FUNCTION_BLOCK FB_MotionAxisDS402NC IMPLEMENTS I_MotionAxis
VAR_INPUT
END_VAR
VAR_OUTPUT
END_VAR
VAR
    {attribute 'no_copy'}
    AxisRef : REFERENCE TO AXIS_REF;
    iMotionAxisCommon : I_MotionAxisCommon;
    // NC Blocks
    fbSetPos		:	MC_SetPosition;
     bClearPositionLag : BOOL := TRUE;

    // create a property for some of these
    bExecMove			: BOOL;
    bExecHome			: BOOL;
    bPosGoal			: BOOL;
    bNegGoal			: BOOL;
    bNewMoveReq			: BOOL;
    bHomingBusy			: BOOL;
    bHomingDone			: BOOL;
    bPrepareDisable		: BOOL;
    bMoveDone			: BOOL;
    bMoveBusy			: BOOL;
    bHalted				: BOOL;
    bAborted			: BOOL;
    bStopped			: BOOL;
    bOperational		: BOOL;
    bServoOffTrans		: BOOL;
    bServoOnTrans 		: BOOL;
    bServoOffMode		: BOOL ;
    bServoOnMode		: BOOL;
    bDiscreteInit		: BOOL;
    bDiscreteMotionAct  : BOOL;
    bServoOffparamsSet  : BOOL;
    bServoOffparamsSetDone : BOOL;
    bLimOverride				: BOOL;
    bPositionHolding		: BOOL;
    bError				: BOOL:=FALSE;
    bErrorStop			: BOOL;
    // use this for motion time axis states
    bExecute			: BOOL;
    // This prevent unexpected logical 1 on stMotionStage.bExecute
    nErrorId			: UDINT:=0;
    sLocalErrorMessage	: STRING;
    nPiezoErrorCode		: UDINT;
    // Save abd restore encoder value
    bInit				: BOOL;
    bLoad				: BOOL;
    bEncError			: BOOL;
    bSaveDone			: BOOL;
    bAbortDone			: BOOL;
    // axis status -- emulating some NC axis
    bClosedLoopMode		:	BOOL;
    bPositiveDirection	:  	BOOL;
    bNegativeDirection 	:  	BOOL;
    bInTargetPosition 	:  	BOOL;
    bReadErrDone			: 	BOOL;
    bLogReady			: 	BOOL;
    bFault				: 	BOOL;
    bDiscreteMotion 	:  	BOOL;
    bContinuousMotion 	:  	BOOL;
    bSlowParamReadTimer	: 	BOOL := TRUE;

    rtHaltedDone	: R_TRIG;
    rtTargetReached	: R_TRIG;
    ftAbortDone: F_TRIG;
    rtFault			: R_TRIG;
    rtHomed			: R_TRIG;
    rtMoveCmdShortcut	: R_TRIG;
    rtHomeCmdShortcut	: R_TRIG;
    rtEnableMode		: R_TRIG;
    rtUserExec			: R_TRIG;
    rtModeChange			: R_TRIG;
    rtTarget		: R_TRIG;
    rtServoOnMode	: R_TRIG;
    rtEnableDrive	: R_TRIG;
    rtServoOnTrans	: R_TRIG;
    rtNotClState 	: R_TRIG;
    rtNotOlState 	: R_TRIG;
    rtNewMoveReq	: R_TRIG;
    rtNewHoldTime	: R_TRIG;
    ftServoOffTrans	: F_TRIG;
    rtServoOffMode	: R_TRIG;
    ftAmsNetId 		: F_TRIG;
    ftExec			: F_TRIG;
    ftErrorSdoRead	: F_TRIG;
    ftEnableDrive	: F_TRIG;
    ftForwardEnabled	: F_TRIG;
    ftBackwardEnabled	: F_TRIG;
    ftServo				: F_TRIG;

    ftSdoStep		: 	F_TRIG;
    ftSdoStepFreq	: 	F_TRIG;
    ftSdoStepAmp	: 	F_TRIG;

    tonSyncHoming 		: TON;
    tonHoldTime			: TON;
    tonServoOffSync		: TON;
    tonSlowParamReadTimer: TON;
    // fast changing paramter timer -- wwe could have used PDO for this params
    // but the Piezo ESC have fixed PDO list.
    tonFastParamReadTimer: TON;
    //bInitiated	: BOOL;
    // Diagnotics data from the drive, mainly Error codes
    tRefreshDelay   : TIME := T#1S;
    nSavedholtime	: UDINT;
    tholtime		: TIME := T#10S;
    // Open Loop Operations
    fbSdoStep		: 	FB_EcCoESdoWrite;
    fbSdoStepFreq	: 	FB_EcCoESdoWrite;
    fbSdoStepAmp	: 	FB_EcCoESdoWrite;

    fbErrorSdoRead			: FB_EcCoESdoRead;
    fbFollowWinSdoRead		: FB_EcCoESdoRead;
    fbSoftLimMaxSdoRead		: FB_EcCoESdoRead;
    fbSoftLimMinSdoRead 	: FB_EcCoESdoRead;
    fbMotorloadSdoRead		: FB_EcCoESdoRead;
    fbGetAmsNetId			: FB_GetLocalAmsNetId;

    sAmsNetId 				: T_AmsNetId;
    nSubIndex  				: BYTE := 0;

      nChanFErrWinIdx		: WORD;
      nChanSoftwareLimIdx	: WORD;
      nChanMotorLoadIdx	: WORD;
    nChanErrorCodeIdx	: WORD;
    nChanOlStepIdx		: WORD;
    nChanOlStepFreqIdx	: WORD;
    nChanOlStepAmpIdx	: WORD;

// NC Exposed Parameters
    bCtrlEnablePosDiffControl     : WORD;
    bEncEnableSoftEndMaxControl   : WORD;
    bEncEnableSoftEndMinControl   : WORD;
    fAccelerationMax              : LREAL;
    fCtrlPosDiffMax               : LREAL;
    fCtrlPosDiffMaxTime           : LREAL;
    fDecelerationMax              : LREAL;
    fEncSoftEndMax                : LREAL;
    fEncSoftEndMin                : LREAL;
    fVeloMaximum                  : LREAL;
    fEncOffset               	  : LREAL;
    fEncScaleFactorInternal       : LREAL;
END_VAR


VAR CONSTANT

    nMotorLoadbase		: WORD := 16#200D;
    nSoftLimBase		: WORD := 16#200e;
    nHomeOffsetBase		: WORD := 16#607C;
    nHomingSpeedBase	: WORD := 16#6099;
    nhomingAccBase		: WORD := 16#609a;
    nErrorCodeBase		: WORD := 16#603f;
    nFErrWinBase		: WORD := 16#6065;
    nOlStepBase			: WORD := 16#2022;
    nOlStepAmpBase		: WORD := 16#2023;
    nOlStepFreqBase		: WORD := 16#2024;
    // this true for SmartAct MCS2 and E-727.
    nChanOfsBase		: WORD := 16#800;
    // DS 402 Motor encoder defective code : this is needed for save and restore.
    nEncErrorCode		: WORD := 16#7300;
END_VAR

{warning 'Add method implementation '}
METHOD CalibrateEncValue
END_METHOD

PROPERTY ControlWord : UINT
GET
END_GET
SET
END_SET
END_PROPERTY

METHOD CyclicCalls
END_METHOD

PROPERTY EncOffset : LREAL
GET
EncOffset := fEncOffset;
END_GET
SET
fEncOffset := EncOffset;
END_SET
END_PROPERTY

{warning 'Add method implementation '}
METHOD EncSaveRestore
END_METHOD

PROPERTY Error : BOOL
GET
Error := bError;
END_GET
SET
bError := Error;
END_SET
END_PROPERTY

PROPERTY ErrorCode : UDINT
GET
ErrorCode := nErrorId;
END_GET
SET
nErrorId := ErrorCode;
END_SET
END_PROPERTY

//FB_Init is always available implicitly and it is used primarily for initialization.
//The return value is not evaluated. For a specific influence, you can also declare the
//methods explicitly and provide additional code there with the standard initialization
//code. You can evaluate the return value.
METHOD FB_Init: BOOL
VAR_INPUT
    bInitRetains: BOOL; // TRUE: the retain variables are initialized (reset warm / reset cold)
    bInCopyCode: BOOL;  // TRUE: the instance will be copied to the copy code afterward (online change)
    AxisReference : REFERENCE TO AXIS_REF;
    //iMotionAxisCommon : I_MotionAxisCommon;
END_VAR
AxisRef REF= AxisReference;
//iMotionAxisCommon := iMotionAxisCommon;
END_METHOD

{warning 'Add method implementation '}
METHOD GearIn
END_METHOD

{warning 'Add method implementation '}
METHOD GearOut
END_METHOD

{warning 'Add method implementation '}
METHOD GetAxisRef : REFERENCE TO AXIS_REF
END_METHOD

{warning 'Add method implementation '}
METHOD GetPowerOverride : LREAL
END_METHOD

{warning 'Add method implementation '}
METHOD Halt
VAR_INPUT
    Deceleration	: LREAL := 0.0;
    Jerk	: LREAL := 0.0;
    BufferMode	: MC_BufferMode := .MC_BufferMode.MC_Aborting;
END_VAR
VAR_OUTPUT
    Done	: BOOL;
    Busy	: BOOL;
    Active	: BOOL;
    CommandAborted	: BOOL;
    Error	: BOOL;
    ErrorID	: UDINT;
    ErrorStr	: T_MaxString;
END_VAR
END_METHOD

{warning 'Add property implementation'}
PROPERTY HaltBusy : BOOL
GET
END_GET
END_PROPERTY

{warning 'Add property implementation'}
PROPERTY HaltDone : BOOL
GET
END_GET
END_PROPERTY

{warning 'Add property implementation'}
PROPERTY HaltError : BOOL
GET
END_GET
END_PROPERTY

{warning 'Add property implementation'}
PROPERTY HaltErrorID : UDINT
GET
END_GET
END_PROPERTY

METHOD Home
//
// tonSyncHoming(PT:=T#500MS);
// (* IMPORTANT: Homing options and parameters must be configured either via the COE online tab or via the service tool *)
// CASE eHomingState OF
//     E_DS402Homing.INIT_HOMING :;
// 		rtModeChange (CLK:=(THIS^.ModeOfOperationDisplay = E_DS402OpMode.HOMING));
//         IF rtModeChange.Q THEN
// 			tonSyncHoming.IN := TRUE;
//             stPiezoStage.nPiezoDriveControl.4:=TRUE;
//         END_IF
// 		IF tonSyncHoming.Q THEN
// 			eHomingState:=E_DS402Homing.HOMING_IN_PROGRESS;
// 		END_IF
//     E_DS402Homing.HOMING_IN_PROGRESS:
//         IF NOT stPiezoStage.stPiezoDriveStatus.TargetReached
//            AND NOT stPiezoStage.stPiezoDriveStatus.Bit13_OpModeSpecific THEN
//                 HomingBusy:=TRUE;
//                 HomeDone:=FALSE;
//
//         // Interrupted
//         ELSIF Stopped AND stPiezoStage.bHalt THEN
//             eHomingState:=E_DS402Homing.HOMING_INTERRUPTED;
//
// 		// Genral Motion error i.e Following error ?
// 		ELSIF stPiezoStage.stPiezoDriveStatus.Bit13_OpModeSpecific THEN
// 			eHomingState:=E_DS402Homing.HOMING_ERROR;
//
//         // Reached
//         ELSIF stPiezoStage.stPiezoDriveStatus.TargetReached
//             AND stPiezoStage.stPiezoDriveStatus.Bit12_OpModeSpecific
//             AND NOT stPiezoStage.stPiezoDriveStatus.Bit13_OpModeSpecific THEN
//             eHomingState:=E_DS402Homing.HOMING_ATTAINED;
//         END_IF
//
//
//     E_DS402Homing.HOMING_INTERRUPTED :;
//         HomingBusy:=FALSE;
//         HomeDone:=FALSE;
// 		Halted := TRUE;
// 		McAxisState:= MC_AxisStates.MC_AXISSTATE_STOPPING;
//
//     E_DS402Homing.HOMING_ATTAINED:;
//         HomingBusy:=FALSE;
// 		tonSyncHoming.IN := FALSE;
// 		tonHoldTime.IN := TRUE;
// 		eHomingState:=E_DS402Homing.HOMING_DONE;
//
//     E_DS402Homing.HOMING_DONE:;
// 		//prepare next move
// 		IF NOT THIS^.PositionHolding THEN
// 			HomeDone:=TRUE;
// 			stPiezoStage.fPosition:=0.0;
// 			fbSetPos.Position := stPiezoStage.fPosition;
// 			fbSetPos.Execute := HomeDone;
// 			IF fbSetPos.bError THEN
// 				eHomingState:=E_DS402Homing.HOMING_ERROR;
// 			ELSE
// 				IF (fbSetPos.bDone) THEN
// 					fbSetPos.Execute := FALSE;
// 				END_IF
// 			END_IF
// 			PositionHolding := TRUE;
// 			stPiezoStage.nPiezoDriveControl.4:=FALSE;
// 		END_IF
//
//
//     E_DS402Homing.HOMING_ERROR :;
// 		Error:= TRUE;
// 		HomeDone:=FALSE;
// 		HomingBusy:= FALSE;
// 		IF fbSetPos.nErrorId <> 0 THEN
// 		// set an Error flag home, homing actually does sdo read on ErrorCode object
// 			ErrorCode := fbSetPos.nErrorId;
// 		ELSE
// 			McAxisState:=MC_AxisStates.MC_AXISSTATE_ERRORSTOP;
// 		END_IF
//
// END_CASE
//
// fbSetPos.Options.ClearPositionLag:= bClearPositionLag;
// fbSetPos( Axis:= stPiezoStage.Axis  );
END_METHOD

{warning 'Add property implementation'}
PROPERTY HomeDone : BOOL
GET
END_GET
SET
END_SET
END_PROPERTY

{warning 'Add property implementation'}
PROPERTY HomingBusy : BOOL
GET
END_GET
SET
END_SET
END_PROPERTY

{warning 'Add property implementation'}
PROPERTY MeasuredAcceleration : LREAL
GET
END_GET
END_PROPERTY

{warning 'Add property implementation'}
PROPERTY MeasuredPosition : LREAL
GET
END_GET
END_PROPERTY

{warning 'Add property implementation'}
PROPERTY MeasuredVelocity : LREAL
GET
END_GET
END_PROPERTY

PROPERTY ModeOfOperation : BOOL
GET
END_GET
SET
END_SET
END_PROPERTY

PROPERTY ModeOfOperationDisplay : INT
GET
END_GET
SET
END_SET
END_PROPERTY

{warning 'Add method implementation '}
METHOD MoveAbsolute
VAR_INPUT
    Position	: LREAL;
    Velocity	: LREAL;
    Acceleration	: LREAL := 0.0;
    Deceleration	: LREAL := 0.0;
    Jerk	: LREAL := 0.0;
    BufferMode	: MC_BufferMode := .MC_BufferMode.MC_Aborting;
END_VAR
VAR_OUTPUT
    Done	: BOOL;
    Busy	: BOOL;
    Active	: BOOL;
    CommandAborted	: BOOL;
    Error	: BOOL;
    ErrorID	: UDINT;
    ErrorStr	: T_MaxString;
END_VAR
END_METHOD

{warning 'Add property implementation'}
PROPERTY MoveAbsoluteBusy : BOOL
GET
END_GET
END_PROPERTY

{warning 'Add property implementation'}
PROPERTY MoveAbsoluteDone : BOOL
GET
END_GET
END_PROPERTY

{warning 'Add property implementation'}
PROPERTY MoveAbsoluteError : BOOL
GET
END_GET
END_PROPERTY

{warning 'Add property implementation'}
PROPERTY MoveAbsoluteErrorID : UDINT
GET
END_GET
END_PROPERTY

{warning 'Add property implementation'}
PROPERTY MoveAbsoluteTargetAcceleration : LREAL
GET
END_GET
END_PROPERTY

{warning 'Add property implementation'}
PROPERTY MoveAbsoluteTargetDeceleration : LREAL
GET
END_GET
END_PROPERTY

{warning 'Add property implementation'}
PROPERTY MoveAbsoluteTargetJerk : LREAL
GET
END_GET
END_PROPERTY

{warning 'Add property implementation'}
PROPERTY MoveAbsoluteTargetPosition : LREAL
GET
END_GET
END_PROPERTY

{warning 'Add property implementation'}
PROPERTY MoveAbsoluteTargetVelocity : LREAL
GET
END_GET
END_PROPERTY

{warning 'Add property implementation'}
PROPERTY MoveBusy : BOOL
GET
END_GET
SET
END_SET
END_PROPERTY

{warning 'Add property implementation'}
PROPERTY MoveDone : BOOL
GET
END_GET
SET
END_SET
END_PROPERTY

{warning 'Add property implementation'}
PROPERTY NegativeMotionIsEnabled : BOOL
GET
END_GET
END_PROPERTY

PROPERTY PositionHolding : BOOL
GET
END_GET
SET
END_SET
END_PROPERTY

{warning 'Add property implementation'}
PROPERTY PositiveMotionIsEnabled : BOOL
GET
END_GET
END_PROPERTY

METHOD Power
VAR_INPUT
    Enable	: BOOL;
    Enable_Positive	: BOOL;
    Enable_Negative	: BOOL;
    (* in percent from 0 to 100 *)
    Override	: LREAL := 100.0;
    BufferMode	: MC_BufferMode := .MC_BufferMode.MC_Aborting;
END_VAR
VAR_OUTPUT
    Status	: BOOL;
    Busy	: BOOL;
    Active	: BOOL;
    Error	: BOOL;
    ErrorID	: UDINT;
    ErrorStr	: T_MaxString;
END_VAR
END_METHOD

{warning 'Add property implementation'}
PROPERTY PowerError : BOOL
GET
END_GET
END_PROPERTY

{warning 'Add property implementation'}
PROPERTY PowerErrorID : UDINT
GET
END_GET
END_PROPERTY

{warning 'Add property implementation'}
PROPERTY PowerIsEnabled : BOOL
GET
END_GET
END_PROPERTY

{warning 'Add property implementation'}
PROPERTY PowerOverride : LREAL
GET
END_GET
END_PROPERTY

PROPERTY PowerStatus : BOOL
GET
END_GET
END_PROPERTY

{warning 'Add method implementation '}
METHOD Reset
VAR_OUTPUT
    Done	: BOOL;
    Busy	: BOOL;
    Error	: BOOL;
    ErrorID	: UDINT;
    ErrorStr	: T_MaxString;
END_VAR
END_METHOD

{warning 'Add property implementation'}
PROPERTY SetpointAcceleration : LREAL
GET
END_GET
END_PROPERTY

{warning 'Add property implementation'}
PROPERTY SetpointJerk : LREAL
GET
END_GET
END_PROPERTY

{warning 'Add property implementation'}
PROPERTY SetpointPosition : LREAL
GET
END_GET
END_PROPERTY

{warning 'Add property implementation'}
PROPERTY SetpointVelocity : LREAL
GET
END_GET
END_PROPERTY

{warning 'Add method implementation '}
METHOD SetPowerOverride
VAR_INPUT
    (* in percent from 0 to 100 *)
    Override	: LREAL;
END_VAR
VAR_OUTPUT
    Status	: BOOL;
    Busy	: BOOL;
    Active	: BOOL;
    Error	: BOOL;
    ErrorID	: UDINT;
    ErrorStr	: T_MaxString;
END_VAR
END_METHOD

END_FUNCTION_BLOCK

(* stored: Version 1.1.0.1
   POU FB_MotionAxisDS402NC: Id {c65bcaa5-32c2-4ba1-a44e-f37d90d611d0}, SpecialFunc None
   Method CalibrateEncValue: Id {91970a26-c709-4b22-9267-b0d1667fe522}
   Property ControlWord: Id {2e23514f-1ff8-4e7d-ba07-c83a3406e12d}
   Get Get: Id {d1d98f73-4ffe-4c5e-ac5b-39dd2029d583}
   Set Set: Id {7fe4a318-1fd6-4879-9b09-7166eef3accc}
   Method CyclicCalls: Id {4817919d-5e20-4c69-8186-0bdf3efe567b}
   Property EncOffset: Id {eb27fba9-5a73-44b3-af11-96a7e15e3ee9}
   Get Get: Id {4f5f199f-c50e-4b22-b7ed-6508a6417ac4}
   Set Set: Id {f81e3843-bcab-4cad-9e8e-d6f853087f87}
   Method EncSaveRestore: Id {395cb6b1-30cf-4c08-973a-ea5683a4aacb}
   Property Error: Id {6591e605-cd47-41e1-b465-f220aaf35b56}
   Get Get: Id {83c61458-bc47-4a5e-a9b2-bc79b90aa45e}
   Set Set: Id {ced43cf6-7634-420d-9841-a2c3186f3ec9}
   Property ErrorCode: Id {e4677a0d-4413-43f2-9c1c-22656f92edde}
   Get Get: Id {dd065214-6bd8-4f8e-aaae-f102862fe903}
   Set Set: Id {a96e7f86-e0ce-40c9-b81e-a4857450ab14}
   Method FB_Init: Id {3c6b89cf-6335-421f-bc49-43ad02ddd5d0}
   Method GearIn: Id {f2f47c3c-7d99-4ce3-b227-d63c7dadbcd1}
   Method GearOut: Id {df7b12cb-8329-492b-be94-64270ee0b5d3}
   Method GetAxisRef: Id {4c207fcd-ec74-4a2e-ba86-459e92aca7f0}
   Method GetPowerOverride: Id {baaece9b-c9ed-489a-91a6-6084d0b1301b}
   Method Halt: Id {b6a8e12d-141b-4b04-b9a3-63a5a6a53059}
   Property HaltBusy: Id {6de0810c-191e-4226-bd42-c87c979bb175}
   Get Get: Id {d49b1f45-1fdf-4987-913a-622876a70ea8}
   Property HaltDone: Id {a8f5b39a-39b9-4a5b-ad34-4985140fd6f3}
   Get Get: Id {c7f2d09e-21b3-40ba-a673-33daea3f18eb}
   Property HaltError: Id {2768033b-365c-4b0f-930b-fb1bc259fcf2}
   Get Get: Id {4cba867e-6440-4471-83ba-4d04bff8bddf}
   Property HaltErrorID: Id {529176ba-5239-45de-acf8-647c49afbae5}
   Get Get: Id {628ea864-33f6-43f6-8f24-83692e88db69}
   Method Home: Id {70bd90c9-eebc-4f8a-a8ba-43919335ed26}
   Property HomeDone: Id {3f03d77b-7aea-46cf-b024-61ea35080b25}
   Get Get: Id {25d464c0-bb5a-4130-86d9-11dd9c72a9ce}
   Set Set: Id {e5508470-c502-4410-bb85-a928cda5c3a3}
   Property HomingBusy: Id {73613f6b-5360-47c4-a9ca-b2b51b8e5224}
   Get Get: Id {21f2fba0-7289-43ea-9a84-75045f357048}
   Set Set: Id {2c2e2af5-2fee-46fd-b099-50f87b0689fc}
   Property MeasuredAcceleration: Id {e265c786-9035-4ea9-82fe-efff9985ed1b}
   Get Get: Id {405282c6-1f48-4d0b-9ca0-a1359e4ad562}
   Property MeasuredPosition: Id {210ba193-d721-4b65-bd1d-f2c43e4f1098}
   Get Get: Id {ea0c0a20-155f-480f-b77a-543c70a9ce7c}
   Property MeasuredVelocity: Id {cc7e62a9-ad83-4971-a6af-2ec0a8bfdfc3}
   Get Get: Id {7e3270c1-6958-4385-8fe5-a7f14d3aeafc}
   Property ModeOfOperation: Id {875d8e8c-6833-41bc-9ba1-506b540ec8bd}
   Get Get: Id {56d86dbd-488d-4d81-8fba-585be7d2afb4}
   Set Set: Id {cb4afb24-f6a8-483d-9128-b2270706924c}
   Property ModeOfOperationDisplay: Id {025cb625-ad11-4c51-9d0f-d907911a35f1}
   Get Get: Id {246a8b29-e645-4a6c-ba23-adb92ac595af}
   Set Set: Id {66c00ddb-4deb-4f26-b4ae-ee600494a340}
   Method MoveAbsolute: Id {6b50c75c-030a-4b3c-9a0b-c342bc66e047}
   Property MoveAbsoluteBusy: Id {2cd6cbfa-43df-4b87-bc54-2038020ebf9b}
   Get Get: Id {b6e2b46f-30ca-4446-92b6-ee2b61e9f9b2}
   Property MoveAbsoluteDone: Id {943f432d-764c-4ecb-a2a2-cb12fcf0605e}
   Get Get: Id {f8486990-9e49-4836-aeaf-28e8593a1573}
   Property MoveAbsoluteError: Id {cf626fd1-69d1-4b24-bf39-eb2bb0e6a669}
   Get Get: Id {cd3b4f88-1fc9-479a-a785-870d96087ddf}
   Property MoveAbsoluteErrorID: Id {66a0e8fd-8446-42d5-8dc1-d21194658885}
   Get Get: Id {06ebca53-388c-4ee1-8791-6f2d219ed147}
   Property MoveAbsoluteTargetAcceleration: Id {85a7ce31-e422-4d55-815b-75f6f2eddb95}
   Get Get: Id {86dfc7b8-790f-4832-9018-cbf0f297986f}
   Property MoveAbsoluteTargetDeceleration: Id {0e4ef2c7-4d34-41bb-b03d-118b7f0b03e9}
   Get Get: Id {37121560-1d7e-4942-bc92-21680601bbc3}
   Property MoveAbsoluteTargetJerk: Id {8119e403-1deb-4a90-bedb-4b1dcfe12cd6}
   Get Get: Id {97349205-8d90-4980-b021-ce4ef7c014b6}
   Property MoveAbsoluteTargetPosition: Id {e1d6496d-5008-43ee-ae2c-af333785de71}
   Get Get: Id {dd8957fc-2f6f-457e-8c95-7815964cb472}
   Property MoveAbsoluteTargetVelocity: Id {4df382a2-3116-4e7b-be1e-d14c3031819d}
   Get Get: Id {e2a6dfe8-fb2a-46a4-8e5f-3597e2316671}
   Property MoveBusy: Id {a9290b1a-1668-4dfa-bd5e-cc7e81c7e750}
   Get Get: Id {3ae4cec8-f3fd-4679-afb0-a63fd3e072cd}
   Set Set: Id {cdaaf44f-f988-4d4f-9218-530b04a36f8c}
   Property MoveDone: Id {9e1531a1-e6a0-4a66-9f95-ebc283cd5a15}
   Get Get: Id {dab091a5-ff32-461f-bacf-c1719e662e8b}
   Set Set: Id {220287e4-3692-4ee3-b73d-897a41576574}
   Property NegativeMotionIsEnabled: Id {c419136a-7e67-4072-b836-78cc8c7dca74}
   Get Get: Id {fa9d6d62-bb9b-4692-8628-c509a0f38156}
   Property PositionHolding: Id {4d252e80-92d2-459f-82bc-7e889c788733}
   Get Get: Id {8d3dc6eb-61b9-42e5-b787-b381bdd2aa3a}
   Set Set: Id {4c2c329c-0ff8-4545-9da1-65a502c3f8b9}
   Property PositiveMotionIsEnabled: Id {f4210734-bd88-49db-a085-cf2cc3ddc720}
   Get Get: Id {881e0050-033c-4af3-9389-3c745f0a9b23}
   Method Power: Id {dd25e964-0517-40f5-924c-4964ca24fa0f}
   Property PowerError: Id {b157fef6-ae05-49ee-b05a-7231ade2f25f}
   Get Get: Id {4dd46f48-26c6-4cf3-b258-858bb12ab4fd}
   Property PowerErrorID: Id {b1c1fc39-4291-4107-94b8-9ae5e59e6ef1}
   Get Get: Id {bb948010-4f02-4aac-a3ea-658089f48b76}
   Property PowerIsEnabled: Id {f1bac38f-a6f1-4fbe-879b-b55cde1ce210}
   Get Get: Id {ab94d513-cd6f-4f9a-b9b2-4020fd45d543}
   Property PowerOverride: Id {7e5d31ab-4b0b-4773-8fab-26ca827e9af2}
   Get Get: Id {9e06fe3b-9c00-4d49-b81b-c0082dbed8fd}
   Property PowerStatus: Id {a1fcac09-eaa5-4dd8-8dbc-d1d1f1c7685d}
   Get Get: Id {2960272a-335f-4434-a3c9-59af96bed5c2}
   Method Reset: Id {a6bfedcd-09ad-4e2e-b0fb-fb5b66d37a7f}
   Property SetpointAcceleration: Id {35df09f7-af10-412c-b5b8-cd15f520d684}
   Get Get: Id {94f09d03-01ad-4f68-9164-4773b797edee}
   Property SetpointJerk: Id {b378fa45-cce4-4de8-84b1-72661da9d428}
   Get Get: Id {dbb8889c-77c4-4f80-81be-834a84700b59}
   Property SetpointPosition: Id {c2596662-270a-4759-9e67-ef75493ff811}
   Get Get: Id {1ca53cc7-289e-444a-afa9-57df6575a7b3}
   Property SetpointVelocity: Id {c430ed88-ac57-4c22-ba59-69ce5d060837}
   Get Get: Id {9c0b191a-47f4-41c3-bf5d-c2be323f98ea}
   Method SetPowerOverride: Id {f5197579-0377-4093-b3b0-a7c948ff579a} *)
